Fanuc KAREL source: kb00002.KL

PROGRAM KB00002
%NOLOCKGROUP
VAR
P1:INTEGER;RESULT:INTEGER
BEGIN
--
P1=1
RESULT=ABS(P1)
END KB00002
